// TIA Portal V19 export
DATA_BLOCK "Interface"   // DB18
{ S7_Optimized_Access := 'TRUE' }
// stored: MemoryReserve 100
   VAR
      LT1_ScaledInput : Real;
      LC1_ControllerOuput : Real;
      LC1_ExtSp : Real := 2.5;
      CV2_ExpSp : Real := 20.0;
      "101CV1_Open" : Bool;
   END_VAR
BEGIN
END_DATA_BLOCK
